FUNCTION_BLOCK PUBLIC FB_Soldering EXTENDS FB_Sequence
VAR_INPUT
END_VAR
VAR_OUTPUT
END_VAR
VAR
END_VAR

SUPER^.Main();
CASE m_SequenceNumber OF
	SequenceStartNamesStart:
		StartDelaySetTime(T#5S);
		IF m_Delay.Q THEN
			SetSequence(SolderingSequenceStep11);
		END_IF
		
	SolderingSequenceStep11:
		StartDelaySetTime(T#5S);
		IF m_Delay.Q THEN
			SetSequence(SolderingSequenceStep12);
		END_IF
	SolderingSequenceStep12:
		StartDelaySetTime(T#5S);
		IF m_Delay.Q THEN
			Done();
		END_IF
	
END_CASE

END_FUNCTION_BLOCK

(* stored: Version 1.1.0.1, ProductVersion 3.1.0.36
   POU FB_Soldering: Id {7c5b309b-ddd2-4dc2-9501-bbf31ea7886e}, SpecialFunc None *)
